FUNCTION_BLOCK RefeedingConveyor EXTENDS Conveyor
VAR_INPUT
END_VAR
VAR_OUTPUT
END_VAR
VAR
	//Sensors
	m_PresencesensorStart : PresenceSensor;
	m_PresencesensorEnd : PresenceSensor;
	
	//Pusher
	m_Switch : Switch;
END_VAR

METHOD METH_Switch_Extend : BOOL
VAR_INPUT
END_VAR
m_Switch.METH_Extend();
END_METHOD

METHOD METH_Switch_Retract : BOOL
VAR_INPUT
END_VAR
m_Switch.METH_Retract();
END_METHOD

PROPERTY WPAtEnd : BOOL
GET
WPAtEnd := m_PresencesensorEnd.Value;
END_GET
END_PROPERTY

PROPERTY WPAtStart : BOOL
GET
WPAtStart := m_PresencesensorStart.Value;
END_GET
END_PROPERTY

END_FUNCTION_BLOCK

(* stored: Version 1.1.0.1, ProductVersion 3.1.4024.4
   POU RefeedingConveyor: Id {fa0aebc4-ed9f-4c35-827c-2b417d6323eb}, SpecialFunc None
   Folder Methods: Id {967d58bb-f7ca-42a9-af62-d96b6810a3c4}
   Folder Properties: Id {dfae9a42-80d3-4208-b526-db2e7c78b19e}
   Method METH_Switch_Extend: Id {f6ff43cd-212b-4b09-bb0d-7a4aad67eb9f}
   Method METH_Switch_Retract: Id {a1cdef5b-49b5-48eb-badd-90d79bc00a40}
   Property WPAtEnd: Id {93b1b83e-a5bf-4f45-a588-281a08b8167f}
   Get Get: Id {ef6fc39e-1c0b-4945-bdc5-0db5ad3573a5}
   Property WPAtStart: Id {478d4f0d-56b9-4a3f-ab25-d23c7f82157c}
   Get Get: Id {91dd4b66-0380-482e-98c0-de0e6e0fda2c} *)
